{attribute 'linkalways'} 
{attribute 'no_explicit_call' := 'This FB is a CLASS and must be accessed using methods or properties'}
{attribute 'enable_dynamic_creation'}
FUNCTION_BLOCK _REAL EXTENDS DatatypeBase
VAR
	localData : REAL;
	activeData : REFERENCE TO REAL REF= localData;
END_VAR

PROPERTY PUBLIC Address : PVOID
GET
Address := ADR(activeData);
END_GET
END_PROPERTY

METHOD PUBLIC ClearReference
VAR_INPUT
END_VAR
activeData REF= localData;
END_METHOD

METHOD PUBLIC Clone : I_Datatype
VAR
    pClone : POINTER TO _REAL;
END_VAR
pClone := __NEW(_REAL(InitialValue := Value));
Clone := pClone^;
END_METHOD

METHOD FB_init : BOOL
VAR_INPUT
	bInitRetains : BOOL; // if TRUE, the retain variables are initialized (warm start / cold start)
	bInCopyCode : BOOL;  // if TRUE, the instance afterwards gets moved into the copy code (online change)
	InitialValue : REAL;
END_VAR
localData := InitialValue;
END_METHOD

PROPERTY PUBLIC IecType : T_MAXSTRING
GET
IecType := 'REAL';
END_GET
END_PROPERTY

METHOD PUBLIC MakeReferenceTo
VAR_INPUT
	ReferenceTarget : REFERENCE TO REAL;
END_VAR
activeData REF= ReferenceTarget;
END_METHOD

METHOD PUBLIC SerializeWith
VAR_INPUT
	Serializer : I_Serializer;
END_VAR
Serializer.AddReal(activeData);
END_METHOD

PROPERTY PUBLIC Size : UDINT
GET
Size := SIZEOF(activeData);
END_GET
END_PROPERTY

METHOD TryDeserializeFrom : BOOL
VAR_INPUT
	Deserializer : I_Deserializer;
END_VAR
TryDeserializeFrom := Deserializer.TryGetReal(activeData);
END_METHOD

METHOD TryMakeReferenceTo : BOOL
VAR_INPUT
	Target : I_Datatype;
END_VAR
VAR
	pTargetData : POINTER TO REAL;
END_VAR
IF NOT (Target.IecType = IecType) THEN
	RETURN;
END_IF

pTargetData := Target.Address;
activeData REF= pTargetData^;
TryMakeReferenceTo := TRUE;
END_METHOD

PROPERTY PUBLIC Value : REAL
GET
Value := activeData;
END_GET
SET
activeData := Value;
END_SET
END_PROPERTY

END_FUNCTION_BLOCK

(* stored: Version 1.1.0.1, ProductVersion 3.1.4024.12
   POU _REAL: Id {cb930906-495d-0445-3653-95714b8382d9}, SpecialFunc None
   Folder Constructor: Id {a8d5b9a2-fd72-07bb-1684-f70d766a0773}
   Property Address: Id {62b17f3f-05c0-0e17-0154-7831daae3411}
   Get Get: Id {73c42311-455e-0545-0f53-7972346c9fad}
   Method ClearReference: Id {e3a00a95-4cd6-06de-0384-556a70add639}
   Method Clone: Id {51e0fa12-a8a6-0872-2530-dee0db6a66b3}
   Method FB_init: Id {ae35ad77-868b-01bd-24a1-53284b0c9912}
   Property IecType: Id {3104f80c-37af-0f3a-2e47-e7c54b55107a}
   Get Get: Id {f299c4a8-b898-010c-397a-0ba7e64cd4d4}
   Method MakeReferenceTo: Id {576e58e7-cd92-04a9-20ff-cfec4fd24097}
   Method SerializeWith: Id {59c0fde9-5886-093b-17d4-1c24e320a6d9}
   Property Size: Id {29fa0728-1dc3-0c00-22d6-0e88c5c3e76b}
   Get Get: Id {eb58c501-44ec-09f7-398a-2227036f063e}
   Method TryDeserializeFrom: Id {83ab23b0-25d6-0d3a-1723-e73b35d764d4}
   Method TryMakeReferenceTo: Id {9821854e-85d8-0c82-0892-3f00c7c33758}
   Property Value: Id {c4c2e369-3ed5-05ea-1904-d25417c9d1d3}
   Get Get: Id {f6f85ac1-ef23-043f-2031-722d8e2b8110}
   Set Set: Id {77197be5-fcef-0873-29e4-0ff781410103} *)
